PROGRAM main
  VAR
    START AT %QX0.1 : BOOL;
    STOP AT %QX0.2 : BOOL;
    SENSOR AT %QX0.3 : BOOL;
    CONVEYOR AT %QX0.0 : BOOL;
    OBJECT_DETECTION AT %QX0.4 : BOOL;
  END_VAR

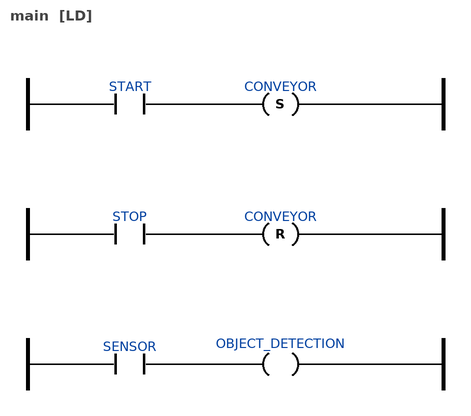
(* LD diagram, written out as Structured Text *)
IF START THEN CONVEYOR := TRUE; END_IF;
IF STOP THEN CONVEYOR := FALSE; END_IF;
OBJECT_DETECTION := SENSOR;
END_PROGRAM
